FUNCTION_BLOCK MetalSaltDosingSensors (* CAT Function Block Type *)
  (* Standard: 61499-2 *)
  (* Version 0.0, 7/9/2026, Schneider Electric, template *)
  PACKAGE SE.Nereda;
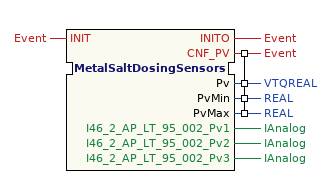
  EVENT_INPUT
    INIT; (* Initializes the symbolic link data destination FB with N (1 <= N <= 16) variables *)
  END_EVENT
  EVENT_OUTPUT
    INITO; (* Initialization Confirm *)
    CNF_PV WITH Pv, PvMin, PvMax; (* Execution confirmation of Pv *)
  END_EVENT
  VAR_OUTPUT
    Pv : VTQREAL; (* Scaled process signal *)
    PvMin : REAL; (* Minimum pv measurement range (in engineering units) *)
    PvMax : REAL; (* Maximun pv measurement range (in engineering units) *)
  END_VAR
  PLUGS
    I46_2_AP_LT_95_002_Pv1 : IAnalog; (* Process value and status interface adapter *)
    I46_2_AP_LT_95_002_Pv2 : IAnalog; (* Process value and status interface adapter *)
    I46_2_AP_LT_95_002_Pv3 : IAnalog; (* Process value and status interface adapter *)
  END_PLUGS
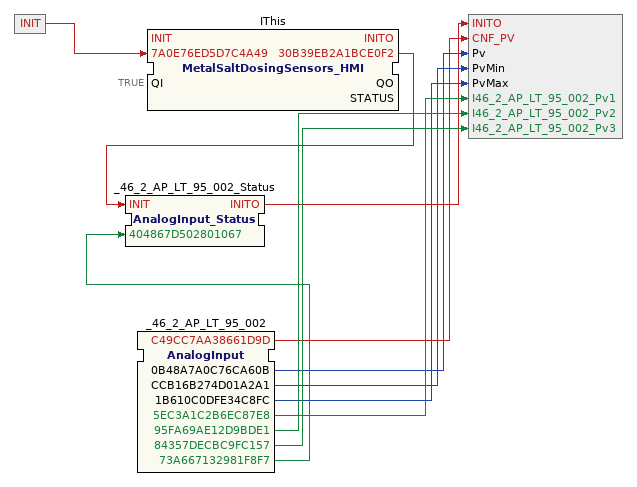
  (* 01 - FUNCTIONNAL INPUT INTERFACE *)
  (* 00 - INITIALIZATION *)
  (* 05 - LOGIC *)
  (* 06 - HMI INTERFACE *)
  (* 02 - FUNCTIONNAL OUTPUT INTERFACE *)
  (* Actuators Status *)
  (* 03 - FIELD INTERFACE *)
  FBS
    _46_2_AP_LT_95_002_Status : AnalogInput_Status;
    _46_2_AP_LT_95_002 : AnalogInput;
    IThis : MetalSaltDosingSensors_HMI(QI := TRUE);
  END_FBS
  EVENT_CONNECTIONS
    IThis.30B39EB2A1BCE0F2 TO _46_2_AP_LT_95_002_Status.INIT;
    _46_2_AP_LT_95_002_Status.INITO TO INITO;
    INIT TO IThis.7A0E76ED5D7C4A49;
    _46_2_AP_LT_95_002.C49CC7AA38661D9D TO CNF_PV;
  END_CONNECTIONS
  DATA_CONNECTIONS
    _46_2_AP_LT_95_002.0B48A7A0C76CA60B TO Pv;
    _46_2_AP_LT_95_002.CCB16B274D01A2A1 TO PvMin;
    _46_2_AP_LT_95_002.1B610C0DFE34C8FC TO PvMax;
  END_CONNECTIONS
  ADAPTER_CONNECTIONS
    _46_2_AP_LT_95_002.5EC3A1C2B6EC87E8 TO I46_2_AP_LT_95_002_Pv1;
    _46_2_AP_LT_95_002.95FA69AE12D9BDE1 TO I46_2_AP_LT_95_002_Pv2;
    _46_2_AP_LT_95_002.84357DECBC9FC157 TO I46_2_AP_LT_95_002_Pv3;
    _46_2_AP_LT_95_002.73A667132981F8F7 TO _46_2_AP_LT_95_002_Status.404867D502801067;
  END_CONNECTIONS
END_FUNCTION_BLOCK
